TYPE (* IEC61131-3, Table 14#5 *)
  (* Standard: 1131-3 *)
  (* Version 0.0, 1/8/2024, Cheyan, Schneider Electric, Template *)
  PACKAGE Main;
  {SET_ATTRIBUTE(nxtDataType, Xek73KlhwgbS2tflgikPNVuxb23cXjysFyjqSNd7amNu/6OF8mveal+6e9ao+YziaWhQUdt602CCVbEazVP+tSuMD2DvtwQSymthxEIuX4jFkNdnAAp4SUU+zeYBFhxj/yXJc1UaeGqRyEeaf6CoJjbC67hEeMPtxZDXZwAKeElK8bxcC8QORMkQM8i2u3yCarWYrZOklUzR774Jl+hKboJVsRrNU/61IzFJ4ioZ1htl/jehx5Fht5HIR5p/oKgmL6UhThn+ty3WZ96iso1N/hkjBrZsGIjw)}
  detailQual : STRUCT
    overflow : BOOL;
    outOfRange : BOOL;
    badReference : BOOL;
    oscillatory : BOOL;
    failure : BOOL;
    oldData : BOOL;
    inconsistent : BOOL;
    inaccurate : BOOL;
  END_STRUCT;
END_TYPE
